// TIA Portal project "QueueOfItems(CT)_V17" (V17)
// Vorlageprojekt für das Buch mit Zielsystem S7-1200

(* hardware
DEVICE "S7-1200-Station_1"  S7-1200 Station
   slot 0: "Baugruppenträger_0"  Rack  V1.0
   slot 1: "PLC_1"  CPU 1211C DC/DC/DC  6ES7 211-1AE40-0XB0  V4.1
DEVICE "HMI_1"  TP700 Comfort
   slot 0: "HMI_1"  TP700 Comfort  6AV2 124-0GC01-0AX0  17.0.0.0
   slot 1: "HMI_RT_1"  TP700 Comfort  6AV2 124-0GC01-0AX0  17.0.0.0
   slot 5: "HMI_1.IE_CP_1"  PROFINET Interface  17.0.0.0
      slot 1: "PROFINET Interface_1"  PROFINET Interface
         slot 1: "Port_1"  Port
         slot 2: "Port_2"  Port
   slot 7: "HMI_1.MPI/DP_CP_1"  MPI/DP Interface  17.0.0.0
*)

// ===== PLC "PLC_1"  CPU 1211C DC/DC/DC =====

VAR_GLOBAL   // PLC tag table "Standard-Variablentabelle"
   "Tag_1" AT %A0.0 : Bool;
   "Tag_2" AT %E0.0 : Bool;
   "Tag_3" AT %E0.1 : Bool;
END_VAR

VAR_GLOBAL   // PLC tag table "Inputs"
   "AtEntrySensor" AT %I10.0 : Bool;
   "AtExitSensor" AT %I10.1 : Bool;
   "ItemReady" AT %I10.2 : Bool;
   "FacoryIORunning" AT %I10.3 : Bool;
END_VAR

VAR_GLOBAL   // PLC tag table "outputs"
   "BufferConvoyer" AT %Q10.0 : Bool;
   "Emitter" AT %Q10.1 : Bool;
   "EntryConvoyer" AT %Q10.2 : Bool;
   "Remover" AT %Q10.3 : Bool;
END_VAR

DATA_BLOCK "Block_1_DB"   // DB2
{ S7_Optimized_Access := 'TRUE' }
VERSION : 0.1
// stored: InstanceOfName Block_1
"Block_1"
BEGIN
END_DATA_BLOCK

DATA_BLOCK "HMI_DB"   // DB9
{ S7_Optimized_Access := 'TRUE' }
VERSION : 0.1
   VAR
      ResetButton : Bool;
      Manual : Bool;
      Auto : Bool;
      ItemReadySensor : Bool;
      AtEntrySensor : Bool;
      AtExitSensor : Bool;
      EntryConvoyerLed : Bool;
      BufferCOnvoyerLed : Bool;
      ItemReadycounter : SInt;
      AtEntryCounter : SInt;
      FactoryIO : Bool;
      ManualEntryCONV : Bool;
      ManualBufferCONV : Bool;
      ResetButtonPE : Bool;
      Operation_MODE : String;
      AtExitCounter : SInt;
   END_VAR
BEGIN
END_DATA_BLOCK

// folder: System blocks/Program resources

DATA_BLOCK "Item_Ready_CTU_DB"   // DB3
{ S7_Optimized_Access := 'TRUE' }
AUTHOR : Simatic
FAMILY : IEC
NAME : CNTR
VERSION : 1.0
// stored: InstanceOfName IEC_COUNTER
"IEC_COUNTER"
BEGIN
END_DATA_BLOCK

DATA_BLOCK "At_Entry_CTU_DB"   // DB5
{ S7_Optimized_Access := 'TRUE' }
AUTHOR : Simatic
FAMILY : IEC
NAME : CNTR
VERSION : 1.0
// stored: InstanceOfName IEC_COUNTER
"IEC_COUNTER"
BEGIN
END_DATA_BLOCK

DATA_BLOCK "At_Exit_CTU_DB"   // DB6
{ S7_Optimized_Access := 'TRUE' }
AUTHOR : Simatic
FAMILY : IEC
NAME : CNTR
VERSION : 1.0
// stored: InstanceOfName IEC_COUNTER
"IEC_COUNTER"
BEGIN
END_DATA_BLOCK

// folder: (top level)

FUNCTION_BLOCK "Block_1"   // FB1, SCL
{ S7_Optimized_Access := 'TRUE' }
VERSION : 0.1
   VAR_INPUT
      at_entry_sensor : Bool;
      at_exit_sensor : Bool;
      manual : Bool;
      auto : Bool;
      reset : Bool;
      man_entry_conv_btn_hmi : Bool;
      man_buffer_conv_btn_hmi : Bool;
      item_ready : Bool;
   END_VAR
   VAR_OUTPUT
      entry_convoyer : Bool;
      buffer_convoyer : Bool;
      factoryio_hmi : Bool;
      item_ready_led_hmi : Bool;
      at_entry_sensor_hmi : Bool;
      at_exit_sensor_hmi : Bool;
      entry_convoyer_led_hmi : Bool;
      buffer_convoyer_led_hmi : Bool;
      item_ready_counter_hmi : SInt;
      at_entry_counter_hmi : SInt;
      OperationMode : String;
      at_exit_counter_hmi : SInt;
   END_VAR
   VAR_IN_OUT
      reset_button_pe : Bool;
   END_VAR
   VAR
      StateMachine : SInt := 0;
      item_ready_sm : Bool;
      at_exit_sm : Bool;
      at_entry_pe : Bool;
      at_entry_sm : Bool;
      MaxItems : SInt := 100;
   END_VAR
   VAR RETAIN
      AtEntryCount : SInt;
   END_VAR
   VAR
      AtExitCount : SInt;
      operation_Mode : SInt;
      ItemReadyCount : SInt;
   END_VAR
BEGIN
   IF "FacoryIORunning" THEN

       #factoryio_hmi := TRUE;

       #item_ready_led_hmi := #item_ready;
       #at_entry_sensor_hmi := #at_entry_sensor;
       #at_exit_sensor_hmi := #at_exit_sensor;

       // Edge detection
       "item_ready_R_TRIG_DB"(CLK := #item_ready,
                              Q => #item_ready_sm);

       "At_Entry_F_TRIG_DB"(CLK := #at_entry_sensor,
                            Q => #at_entry_sm);

       "At_Entry_R_TRIG_DB"(CLK := #at_entry_sensor,
                            Q => #at_entry_pe);

       "At_Exit_F_TRIG_DB"(CLK := #at_exit_sensor,
                           Q => #at_exit_sm);

       "Reset_R_TRIG_DB"(CLK := #reset,
                         Q => #reset_button_pe);

       // Counters
       "Item_Ready_CTU_DB".CTU(CU := #item_ready_sm,
                               PV := #MaxItems,
                               CV => #ItemReadyCount,
                               R := #reset_button_pe);

       #item_ready_counter_hmi := "Item_Ready_CTU_DB".CV;

       "At_Entry_CTU_DB".CTU(CU := #at_entry_sm,
                             PV := #MaxItems,
                             CV => #AtEntryCount,
                             R := #reset_button_pe);

       #at_entry_counter_hmi := "At_Entry_CTU_DB".CV;

       "At_Exit_CTU_DB".CTU(CU := #at_exit_sm,
                            PV := #MaxItems,
                            CV => #AtExitCount,
                            R := #reset_button_pe);

       #at_exit_counter_hmi := "At_Exit_CTU_DB".CV;

       // Operation Mode Select
       // Reset = highest priority
       IF #reset_button_pe THEN
           #operation_Mode := 2;
       ELSIF #auto THEN
           #operation_Mode := 1;
       ELSIF #manual THEN
           #operation_Mode := 0;
       END_IF;

       // Operation Mode definitions
       // 0 = Manual
       // 1 = Auto  
       // 2 = Reset
       // 3 = Idle (waiting for operator)

       CASE #operation_Mode OF

           0: // Manual Mode
               #OperationMode := 'Manual';

               #entry_convoyer := #man_entry_conv_btn_hmi;
               #buffer_convoyer := #man_buffer_conv_btn_hmi;

           1: // Auto Mode
               #OperationMode := 'Automatique';
               IF #item_ready_sm THEN
                   #entry_convoyer := TRUE;
               END_IF;

               IF #at_entry_pe THEN
                   #buffer_convoyer := TRUE;
               END_IF;

               IF "Item_Ready_CTU_DB".CV = "At_Entry_CTU_DB".CV
                   AND ("Item_Ready_CTU_DB".CV > 0) THEN
                   #entry_convoyer := FALSE;
               END_IF;

               IF "At_Exit_CTU_DB".CV = "At_Entry_CTU_DB".CV
                   AND ("At_Exit_CTU_DB".CV > 0) AND #at_exit_sm THEN
                   #buffer_convoyer := FALSE;
               END_IF;

           2: // Reset
               #OperationMode := 'Reset';

               "Item_Ready_CTU_DB".R := TRUE;
               "At_Entry_CTU_DB".R := TRUE;
               "At_Exit_CTU_DB".R := TRUE;

               #entry_convoyer := FALSE;
               #buffer_convoyer := FALSE;
               #operation_Mode := 3;

           3: // Idle - waiting for operator
               #OperationMode := 'IDLE';
               #reset_button_pe := false;

               "Item_Ready_CTU_DB".R := False;
               "At_Entry_CTU_DB".R := false;
               "At_Exit_CTU_DB".R := false;

               #entry_convoyer := FALSE;
               #buffer_convoyer := FALSE;

       END_CASE;

       // Convoyers LED logic 
       #entry_convoyer_led_hmi := #entry_convoyer;
       #buffer_convoyer_led_hmi := #buffer_convoyer;

   ELSE
       #factoryio_hmi := FALSE;

   END_IF;
END_FUNCTION_BLOCK

FUNCTION "MHJ-PLC-Lab-Function-S71200" : Void   // FC9000, SCL
{ S7_Optimized_Access := 'TRUE' }
VERSION : 0.1
   VAR_TEMP
      rdTimeReturn : Int;
      outputTime : DTL;
      SyncVal : Byte;
      forVal : Int;
      forVal_2 : Int;
      Value : Byte;
   END_VAR
   VAR CONSTANT
      CompVal : Byte := 16#34;
      Value_01 : Byte := 16#11;
      Value_01_DW : DWord := 16#A165_D992;
      Value_02_DW : DWord := 16#58BE_4401;
   END_VAR
BEGIN

   #Value:=PEEK(area := 16#82,
        dbNumber := 0,
        byteOffset := 511);
   #Value := #Value + 1;

   POKE(area := 16#82,
        dbNumber := 0,
        byteOffset := 511,
        value := #Value);

   POKE(area:=16#81,
        dbNumber:=0,
        byteOffset:=1016,
        value:=#Value_01_DW);
   POKE(area := 16#81,
        dbNumber := 0,
        byteOffset := 1020,
        value := #Value_02_DW);

   POKE(area := 16#81,
        dbNumber := 0,
        byteOffset := 511,
        value := B#16#00);

   FOR #forVal := 0 TO 120 DO
       FOR #forVal_2:=0 TO 10 DO
           #rdTimeReturn:=RD_SYS_T(#outputTime);
           #rdTimeReturn := WR_SYS_T(#outputTime);
           #rdTimeReturn := RD_SYS_T(#outputTime);
           #rdTimeReturn := WR_SYS_T(#outputTime);
       END_FOR;
       #SyncVal:= PEEK(area := 16#81,
                      dbNumber := 0,
                      byteOffset := 511);
       IF #SyncVal = #CompVal THEN
          GOTO M_1;
       END_IF;
   END_FOR;
   RETURN;

   M_1:
   POKE(area := 16#81,
        dbNumber := 0,
        byteOffset := 511,
        value := B#16#0);
END_FUNCTION

ORGANIZATION_BLOCK "Main"   // OB1, LAD, ProgramCycle
TITLE = "Main Program Sweep (Cycle)"
{ S7_Optimized_Access := 'TRUE' }
VERSION : 0.1
   VAR_INPUT
      Initial_Call : Bool;   // Initial call of this OB
      Remanence : Bool;   // =True, if remanent data are available
   END_VAR
BEGIN

REGION Network 1: Konnektierungsbaustein für PLC-Lab
   // Im Netzwerk 1 wird der Konnektierungsbaustein für PLC-Lab aufgerufen.
   // Dieser Aufruf darf nicht entfernt werden!
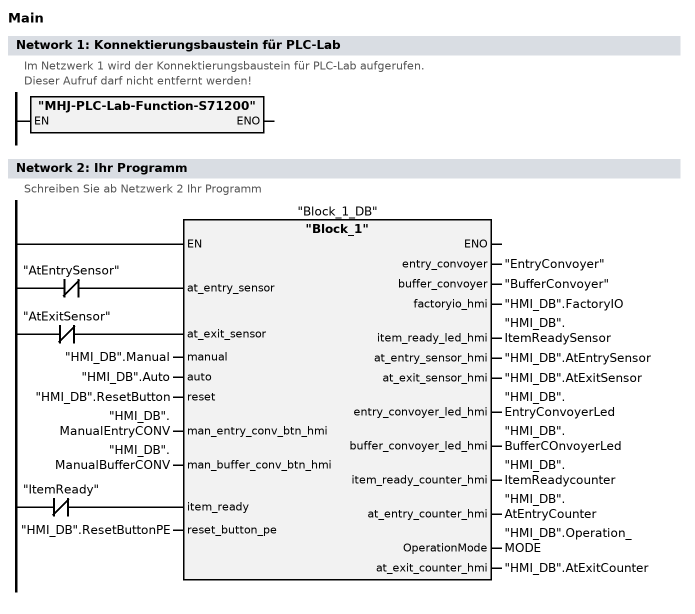
   RUNG wire#powerrail
      "MHJ-PLC-Lab-Function-S71200"()
   END_RUNG
   // the same network as SCL:
   "MHJ-PLC-Lab-Function-S71200"();
END_REGION

REGION Network 2: Ihr Programm
   // Schreiben Sie ab Netzwerk 2 Ihr Programm
   RUNG wire#powerrail
      "Block_1_DB"(at_entry_sensor := wire#w1, at_exit_sensor := wire#w2, item_ready := wire#w3, manual := "HMI_DB".Manual, auto := "HMI_DB".Auto, reset := "HMI_DB".ResetButton, man_entry_conv_btn_hmi := "HMI_DB".ManualEntryCONV, man_buffer_conv_btn_hmi := "HMI_DB".ManualBufferCONV, reset_button_pe := "HMI_DB".ResetButtonPE, entry_convoyer => "EntryConvoyer", buffer_convoyer => "BufferConvoyer", factoryio_hmi => "HMI_DB".FactoryIO, item_ready_led_hmi => "HMI_DB".ItemReadySensor, at_entry_sensor_hmi => "HMI_DB".AtEntrySensor, at_exit_sensor_hmi => "HMI_DB".AtExitSensor, entry_convoyer_led_hmi => "HMI_DB".EntryConvoyerLed, buffer_convoyer_led_hmi => "HMI_DB".BufferCOnvoyerLed, item_ready_counter_hmi => "HMI_DB".ItemReadycounter, at_entry_counter_hmi => "HMI_DB".AtEntryCounter, OperationMode => "HMI_DB".Operation_MODE, at_exit_counter_hmi => "HMI_DB".AtExitCounter)
   END_RUNG
   RUNG wire#powerrail
      I_Contact( "AtEntrySensor" )
   END_RUNG wire#w1
   RUNG wire#powerrail
      I_Contact( "AtExitSensor" )
   END_RUNG wire#w2
   RUNG wire#powerrail
      I_Contact( "ItemReady" )
   END_RUNG wire#w3
   // the same network as SCL:
   "Block_1_DB"(at_entry_sensor := NOT "AtEntrySensor",   // "Block_1"
                at_exit_sensor := NOT "AtExitSensor",
                manual := "HMI_DB".Manual,
                auto := "HMI_DB".Auto,
                reset := "HMI_DB".ResetButton,
                man_entry_conv_btn_hmi := "HMI_DB".ManualEntryCONV,
                man_buffer_conv_btn_hmi := "HMI_DB".ManualBufferCONV,
                item_ready := NOT "ItemReady",
                reset_button_pe := "HMI_DB".ResetButtonPE,
                entry_convoyer => "EntryConvoyer",
                buffer_convoyer => "BufferConvoyer",
                factoryio_hmi => "HMI_DB".FactoryIO,
                item_ready_led_hmi => "HMI_DB".ItemReadySensor,
                at_entry_sensor_hmi => "HMI_DB".AtEntrySensor,
                at_exit_sensor_hmi => "HMI_DB".AtExitSensor,
                entry_convoyer_led_hmi => "HMI_DB".EntryConvoyerLed,
                buffer_convoyer_led_hmi => "HMI_DB".BufferCOnvoyerLed,
                item_ready_counter_hmi => "HMI_DB".ItemReadycounter,
                at_entry_counter_hmi => "HMI_DB".AtEntryCounter,
                OperationMode => "HMI_DB".Operation_MODE,
                at_exit_counter_hmi => "HMI_DB".AtExitCounter);
END_REGION
END_ORGANIZATION_BLOCK

(* ===== HMI "HMI_RT_1" =====
system functions are stored by id; their names below are inferred from use
connection "HMI_Connection_1": ETHERNET, S7_1200_OMS

HMI tags "Default tag table"
   "Tag_ScreenNumber" : UInt, internal
   "HMI_DB_FactoryIO" : Bool = PLC HMI_DB.FactoryIO, 1 s
   "HMI_DB_ItemReadySensor" : Bool = PLC HMI_DB.ItemReadySensor, 1 s
   "HMI_DB_AtEntrySensor" : Bool = PLC HMI_DB.AtEntrySensor, 1 s
   "HMI_DB_AtExitSensor" : Bool = PLC HMI_DB.AtExitSensor, 1 s
   "HMI_DB_EntryConvoyerLed" : Bool = PLC HMI_DB.EntryConvoyerLed, 1 s
   "HMI_DB_BufferCOnvoyerLed" : Bool = PLC HMI_DB.BufferCOnvoyerLed, 1 s
   "HMI_DB_ItemReadycounter" : SInt = PLC HMI_DB.ItemReadycounter, 1 s
   "HMI_DB_AtEntryCounter" : SInt = PLC HMI_DB.AtEntryCounter, 1 s
   "HMI_DB_AtExitCounter" : SInt = PLC HMI_DB.AtExitCounter, 1 s
   "HMI_DB_Auto" : Bool = PLC HMI_DB.Auto, 1 s
   "HMI_DB_Manual" : Bool = PLC HMI_DB.Manual, 1 s
   "HMI_DB_ResetButton" : Bool = PLC HMI_DB.ResetButton, 1 s
   "HMI_DB_Operation_MODE" : String[254] = PLC HMI_DB.Operation_MODE, 1 s
   "HMI_DB_ManualEntryCONV" : Bool = PLC HMI_DB.ManualEntryCONV, 1 s
   "HMI_DB_ManualBufferCONV" : Bool = PLC HMI_DB.ManualBufferCONV, 1 s
   "HMI_DB_ResetButtonPE" : Bool = PLC HMI_DB.ResetButtonPE, 1 s

screen "Root screen" 800x420, template "Template_1"
   on GenerateScreen: SetTag("Tag_ScreenNumber", 1)
   Rectangle "Rectangle_4" at 660,6 size 137x106
      Visibility <- "HMI_DB_Auto"
   Rectangle "Rectangle_3" at 669,3 size 130x211
      Visibility <- "HMI_DB_Manual"
   TextField "HmiScreenItemData_3" at 405,38 size 107x23; Text 'EntryConvoyer'
   TextField "HmiScreenItemData_4" at 510,38 size 122x23; Text 'BufferConvoyer'
   Circle "Circle_6" at 557,15 size 23x23
      Visibility <- "HMI_DB_BufferCOnvoyerLed"
   Circle "Circle_5" at 557,15 size 23x23
      Visibility <- "HMI_DB_BufferCOnvoyerLed"
   Circle "Circle_4" at 441,15 size 23x23
      Visibility <- "HMI_DB_EntryConvoyerLed"
   Circle "Circle_3" at 441,15 size 23x23
      Visibility <- "HMI_DB_EntryConvoyerLed"
   Circle "Circle_2" at 49,15 size 23x23
      Visibility <- "HMI_DB_FactoryIO"
   Circle "Circle_1" at 49,15 size 23x23
      Visibility <- "HMI_DB_FactoryIO"
   TextField "HmiScreenItemData_2" at 1,38 size 110x25; Text 'FactoryIO'
   Circle "Circle_7" at 238,15 size 23x23
      Visibility <- "HMI_DB_AtEntrySensor"
   Circle "Circle_8" at 238,15 size 23x23
      Visibility <- "HMI_DB_AtEntrySensor"
   Circle "Circle_9" at 132,15 size 23x23
      Visibility <- "HMI_DB_ItemReadySensor"
   Circle "Circle_10" at 132,15 size 23x23
      Visibility <- "HMI_DB_ItemReadySensor"
   Circle "Circle_11" at 322,15 size 23x23
      Visibility <- "HMI_DB_AtExitSensor"
   Circle "Circle_12" at 322,15 size 23x23
      Visibility <- "HMI_DB_AtExitSensor"
   TextField "HmiScreenItemData_1" at 89,38 size 107x23; Text 'ItemReady'
   TextField "HmiScreenItemData_5" at 196,38 size 107x23; Text 'AtEntry'
   TextField "HmiScreenItemData_6" at 278,38 size 107x23; Text 'AtExit'
   GraphicView "Graphic view_2" at 38,127 size 300x205; Picture "Graphic_3"
   GraphicView "Graphic view_3" at 336,127 size 300x205; Picture "Graphic_3"
   IOField "I/O field_1" at 35,233 size 50x30; FormatPattern s99
      ProcessValue <- "HMI_DB_ItemReadycounter"
   IOField "I/O field_2" at 313,234 size 50x30; FormatPattern s99
      ProcessValue <- "HMI_DB_AtEntryCounter"
   IOField "I/O field_3" at 601,233 size 48x30; FormatPattern s99
      ProcessValue <- "HMI_DB_AtExitCounter"
   TextField "HmiScreenItemData_7" at 0,264 size 110x25; Text 'ItemReady'
   TextField "HmiScreenItemData_8" at 278,266 size 110x25; Text 'AtEntry'
   TextField "HmiScreenItemData_9" at 567,266 size 110x25; Text 'AtExit'
   TextField "HmiScreenItemData_10" at 0,276 size 110x25; Text 'Counter'
   TextField "HmiScreenItemData_11" at 278,277 size 110x25; Text 'Counter'
   TextField "HmiScreenItemData_12" at 567,277 size 110x25; Text 'Counter'
   Switch "Switch_1" at 681,50 size 94x44; CaptionText 'Switch'; TextOff 'MAN'; TextOn 'AUTO'
      on SwitchOn: SetBit("HMI_DB_Auto"); ResetBit("HMI_DB_Manual")
      on SwitchOff: SetBit("HMI_DB_Manual"); ResetBit("HMI_DB_Auto")
   TextField "Text field_1" at 686,14 size 86x20; Text 'Operation'
   TextField "Text field_2" at 709,30 size 41x20; Text 'Mode'
   Button "Button_1" at 675,127 size 115x32; TextOff 'EntryCONV'
      Visibility <- "HMI_DB_Manual"
      on Press: SetBit("HMI_DB_ManualEntryCONV")
      on Release: ResetBit("HMI_DB_ManualEntryCONV")
   Button "Button_2" at 675,172 size 115x32; TextOff 'BufferCONV'
      Visibility <- "HMI_DB_Manual"
      on Release: SetBit("HMI_DB_ManualBufferCONV")
      on Activate: ResetBit("HMI_DB_ManualBufferCONV")
   TextField "Text field_3" at 675,99 size 131x20; Text 'Manual Entries'
      Visibility <- "HMI_DB_Manual"
   Button "Button_3" at 681,302 size 96x32; TextOff 'Reset'
      on Press: SetBit("HMI_DB_ResetButton")
      on Release: ResetBit("HMI_DB_ResetButton")
   IOField "I/O field_4" at 313,87 size 169x32; FormatPattern ???????????????
      ProcessValue <- "HMI_DB_Operation_MODE"
   TextField "Text field_5" at 120,87 size 173x26; Text 'Operation Mode'
   Circle "Circle_13" at 706,228 size 48x48
      Visibility <- "HMI_DB_ResetButtonPE"
   Circle "Circle_14" at 706,228 size 48x48
      Visibility <- "HMI_DB_ResetButtonPE"

Template "Template_1" 800x420
   Button "Exit" at 720,360 size 78x58; TextOff 'Exit'; PictureOff "ExitRuntime_TP700_Comfort_TR"; PictureOn "ExitRuntime_TP700_Comfort_TR"
      on Release: StopRuntime(0)
   Button "Template_Button" at 640,360 size 78x58; TextOff 'Text'
   Button "Template_Button_1" at 560,360 size 78x58; TextOff 'Text'
   Button "Template_Button_2" at 480,360 size 78x58; TextOff 'Text'
   Button "Template_Button_3" at 400,360 size 78x58; TextOff 'Text'
   Button "Template_Button_4" at 321,360 size 78x58; TextOff 'Text'
   Button "Template_Button_5" at 241,360 size 78x58; TextOff 'Text'
   Button "Template_Button_6" at 161,360 size 78x58; TextOff 'Text'
   Button "Template_Button_7" at 81,360 size 78x58; TextOff 'Text'
   Button "Start screen" at 1,360 size 78x58; TextOff 'Start screen'; PictureOff "NavigateHome_TP700_Comfort_TR"; PictureOn "NavigateHome_TP700_Comfort_TR"
      on Release: ActivateScreen("Root screen", 0)
*)